FUNCTION_BLOCK FB_Auto
VAR_INPUT
END_VAR
VAR_OUTPUT
END_VAR
VAR
END_VAR

END_FUNCTION_BLOCK

(* stored: Version 1.1.0.1, ProductVersion 3.1.4024.13
   POU FB_Auto: Id {f600c05e-242e-4e37-a43b-79e2b5f278fc}, SpecialFunc None *)
